Fanuc KAREL source: NC0090.KL

-- PROVISIONAL review KL for V940-1; original PC SHA256 7678b7e07e84ef13661e2eb628a7e6db1e44701450144df40a58f48f49e1c7ce
-- Incomplete behavior may be omitted. Consult companion uncertainty JSON. Do not deploy.
PROGRAM NC0090
%NOLOCKGROUP
-- UNRESOLVED_LOCAL_POOL 5 cells at code offset 3; source declarations unknown
-- DIRECT_LOCAL_WORD_ACCESS alone does not prove INTEGER, REAL, or BOOLEAN
BEGIN
  -- V9_OWNER_INTERVAL_HINT [23,229),[45,198),[67,167),[89,136); structural only; source/VM held
  -- V9_FOOTER_20_HINT 4 numerical footer links; VM transfer unproved
  -- UNRESOLVED_PC offsets 0-8; opcodes 2B,2C,7B
  -- UNRESOLVED_PC offsets 13-20; opcodes 9D,23
  -- UNRESOLVED_PC offsets 25-38; opcodes 21,9D,57,79
  -- UNRESOLVED_PC offsets 43-60; opcodes 21,40,41,42
  -- UNRESOLVED_PC offsets 65-94; opcodes 9D,23,9E,2E,22,7A
  -- UNRESOLVED_PC offsets 99-116; opcodes 21,2E,59,79
  -- UNRESOLVED_PC offsets 121-134; opcodes 21,9D,57,79
  -- UNRESOLVED_PC offsets 139-156; opcodes 21,40,41,42
  -- UNRESOLVED_PC offsets 161-190; opcodes 9D,23,9E,2E,22,7A
  -- UNRESOLVED_PC offsets 195-212; opcodes 21,2E,59,79
  -- UNRESOLVED_PC offsets 217-230; opcodes 21,9D,57,79
  -- UNRESOLVED_PC offsets 235-252; opcodes 21,40,41,42
  -- UNRESOLVED_PC offsets 257-286; opcodes 9D,23,9E,2E,22,7A
  -- UNRESOLVED_PC offsets 291-308; opcodes 21,2E,59,79
  -- UNRESOLVED_PC offsets 313-326; opcodes 21,9D,57,79
  -- UNRESOLVED_PC offsets 331-348; opcodes 21,40,41,42
  -- UNRESOLVED_PC offsets 353-382; opcodes 9D,23,9E,2E,22,7A
  -- UNRESOLVED_PC offsets 387-404; opcodes 21,2E,59,79
  -- UNRESOLVED_PC offsets 409-422; opcodes 21,9D,57,79
  -- UNRESOLVED_PC offsets 427-444; opcodes 21,40,41,42
  -- UNRESOLVED_PC offsets 449-479; opcodes 21,9D,52,23,7A,40,41,42
  -- UNRESOLVED_PC offsets 484-508; opcodes 21,2E,52,23,7A,43
  -- UNRESOLVED_PC offsets 513-531; opcodes 21,2E,52,23
  -- UNRESOLVED_PC offsets 541-546; opcodes 7A
  -- UNRESOLVED_PC offsets 551-569; opcodes 21,2E,52,23
  -- UNRESOLVED_PC offsets 579-584; opcodes 7A
  -- UNRESOLVED_PC offsets 589-620; opcodes 20,2C,23,7A,40,41,42
  -- UNRESOLVED_PC offsets 625-649; opcodes 21,2E,52,23,7A,43
  -- UNRESOLVED_PC offsets 654-672; opcodes 21,2E,52,23
  -- UNRESOLVED_PC offsets 682-687; opcodes 7A
  -- UNRESOLVED_PC offsets 692-710; opcodes 21,2E,52,23
  -- UNRESOLVED_PC offsets 720-725; opcodes 7A
  -- UNRESOLVED_PC offsets 730-761; opcodes 20,2C,23,7A,40,41,42
  -- UNRESOLVED_PC offsets 766-790; opcodes 21,2E,52,23,7A,43
  -- UNRESOLVED_PC offsets 795-813; opcodes 21,2E,52,23
  -- UNRESOLVED_PC offsets 823-828; opcodes 7A
  -- UNRESOLVED_PC offsets 833-851; opcodes 21,2E,52,23
  -- UNRESOLVED_PC offsets 861-866; opcodes 7A
  -- UNRESOLVED_PC offsets 871-902; opcodes 20,2C,23,7A,40,41,42
  -- UNRESOLVED_PC offsets 907-931; opcodes 21,2E,52,23,7A,43
  -- UNRESOLVED_PC offsets 936-954; opcodes 21,2E,52,23
  -- UNRESOLVED_PC offsets 964-969; opcodes 7A
  -- UNRESOLVED_PC offsets 974-992; opcodes 21,2E,52,23
  -- UNRESOLVED_PC offsets 1002-1007; opcodes 7A
  -- UNRESOLVED_PC offsets 1012-1043; opcodes 20,2C,23,7A,40,41,42
  -- UNRESOLVED_PC offsets 1048-1072; opcodes 21,2E,52,23,7A,43
  -- UNRESOLVED_PC offsets 1077-1095; opcodes 21,2E,52,23
  -- UNRESOLVED_PC offsets 1105-1110; opcodes 7A
  -- UNRESOLVED_PC offsets 1115-1133; opcodes 21,2E,52,23
  -- UNRESOLVED_PC offsets 1143-1147; opcodes 7F
  -- UNRESOLVED_PC offsets 1152-1156; opcodes 27,AA
  -- UNRESOLVED_PC offsets 1161-1165; opcodes 7F
END NC0090
